{attribute 'qualified_only'}
{attribute 'strict'}
TYPE LidStates :
(
	WaitingToStart,LocatingInPlace,PickingAndPlacing,Stop
);
END_TYPE

(* stored: Version 1.1.0.1, ProductVersion 3.1.4024.9
   DUT LidStates: Id {25e30745-b4d0-4d1c-b608-0bbd938cff1c} *)
